(* IEC 61131-3 sources: Industry-PLC-LLM/data/PLCBEAD_repo/PLCBEAD_PLCEmbed-main/PLC-BEAD/Source/GEB/BIT_OF_DWORD, 1 file *)

(* ---- BIT_OF_DWORD.ST ---- *)
FUNCTION BIT_OF_DWORD : BOOL
  VAR_INPUT
    IN : DWORD;
    N : INT;
  END_VAR

  BIT_OF_DWORD := (SHR(IN,N) AND 16#00000001) > 0;
END_FUNCTION

PROGRAM program0
  VAR
    LocalVar0 : DWORD;
    LocalVaR2 : INT;
    LocalVaR1  : BOOL;
    CEIL5_OUT : BOOL;
  END_VAR

  CEIL5_OUT := BIT_OF_DWORD(LocalVar0, LocalVaR2);
  LocalVaR1  := CEIL5_OUT;
END_PROGRAM
